// TIA Portal V18 export
FUNCTION_BLOCK "I_TRIG_int_change"   // FB52, FBD
{ S7_Optimized_Access := 'TRUE' }
VERSION : 0.1
// stored: AutoNumber true, IsIECCheckEnabled false, IsRetainMemResEnabled false, MemoryReserve 100, SetENOAutomatically false, UDAEnableTagReadback false
   VAR_INPUT
      J : Int;
   END_VAR
   VAR_OUTPUT
      C : Bool;
   END_VAR
   VAR
      J_was : Int;
   END_VAR
BEGIN

REGION Network 1
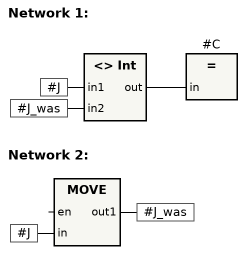
   #C := #J <> #J_was;
END_REGION

REGION Network 2
   #J_was := #J;
END_REGION
END_FUNCTION_BLOCK
